Staubli VAL3: sendJointFbk.pgx

public program sendJointFbk()
  local num l_nRetVal
begin

end
